// TwinCAT 3 PLC project DAS_assignment1_AbhijitDas
// ProgramVersion: 3.1.0.9
// libraries:
//   Standard, * (System)
//   VisuElem3DPath, 3.5.6.0 (System)
//   VisuElemMeter, 3.5.6.0 (System)
//   VisuElems, 3.5.6.10 (System)
//   VisuElemsDateTime, 3.5.6.0 (System)
//   VisuElemsSpecialControls, 3.5.6.0 (System)
//   VisuElemsWinControls, 3.5.6.0 (System)
//   VisuElemTextEditor, 3.5.6.0 (System)
//   visuinputs, 3.5.6.0 (system)
//   VisuNativeControl, 3.5.6.0 (System)
//   Tc2_Standard, * (Beckhoff Automation GmbH)
//   Tc2_System, * (Beckhoff Automation GmbH)
//   Tc3_Interfaces, * (Beckhoff Automation GmbH)
//   Tc3_Module, * (Beckhoff Automation GmbH)
//   VisuDialogs, * (System)
// project tree:
//   / GlobalTextList.TcGTLO, GVL.TcGVL, PlcTask.TcTTO, Visualization Manager.TcVMO (not stored)
//   POUs/ DistStationSensors.TcPOU, DistStationControl.TcPOU, MAIN.TcPOU, TestStationControl.TcPOU, TestStationSensors.TcPOU
//   VISUs/ StationVisualProgram.TcPOU, StationVisual.TcVIS

CONFIGURATION DAS_assignment1_AbhijitDas
    RESOURCE PLC ON TwinCAT3
        TASK PlcTask(INTERVAL := T#10ms, PRIORITY := 20);
        PROGRAM MAIN WITH PlcTask : MAIN;
    END_RESOURCE
END_CONFIGURATION

// ---- GVL.TcGVL
VAR_GLOBAL
	
	
	insertMag: BOOL; (* Variable for inserting Cylinder base in the stack magazine barrel*)
	Check_Mat: BOOL; (* Variable for starting the material checking actuator*)
	H_Meas: BOOL;   (* Variable for starting the height measurement actuator*)
	Testing: BOOL;  (* Variable that is set while the testing station is busy*)
	T_reset: TIME;	(* time to imitate reset value*)
	VisuReset: BOOL := TRUE; (* Variable is used to reset the visualization when reset is pressed*)
	forVisuPos5: BOOL;   (* used for visual only*)
	
	
	(* These variables are all as described in the provided MPS Festo documents*)
	start: BOOL;
	stop: BOOL;
	reset: BOOL;
	Mag: BOOL;
	Mag_back: BOOL := TRUE;
	Mag_front: BOOL;
	Vacuum: BOOL;
	Arm_take: BOOL := TRUE;
	Arm_put: BOOL;
	Mat_sen: BOOL;
	Vacumon: BOOL;
	Vacumoff: BOOL;
	Armleft: BOOL;
	Armright: BOOL;
	Auto: BOOL;
	Automan: BOOL;
	L_START: BOOL;
	L_RESET: BOOL;
	LiftDown: BOOL;
	MatPush: BOOL;
	Slide: BOOL;
	Part_AV: BOOL;
	Lift_Up: BOOL;
	Push_Ba: BOOL;
	Sen_Mat: BOOL;
	LiftUp: BOOL;
	Lift_Down: BOOL := TRUE;
	Work_ok: BOOL := TRUE;
	Follow: BOOL;
	Safety_barrier: BOOL;
	
	
END_VAR

// ---- POUs/MAIN.TcPOU
PROGRAM MAIN
VAR
END_VAR

DistStationSensors();
DistStationControl();
TestStationSensors();
TestStationControl();
StationVisualProgram();

END_PROGRAM

// ---- POUs/DistStationSensors.TcPOU
PROGRAM DistStationSensors
VAR
	StackLimit: WORD := 8; (* Stating the limit of the stack module barrel*)
	null: BOOL; (* set when stack module barrel is empty*)
	Current: WORD ; (* Current number of base/s in the stack module barrel*)
	LimitReached: BOOL; (* set when the stack module barrel is full*)
	counter1: CTUD;  (* counter used to count the number of bases inserted in the barrel*)
	
END_VAR
VAR // added by the converter: edge detectors and wires of the graphical bodies
    _w1, _w2, _w3, _w4 : BOOL;
END_VAR

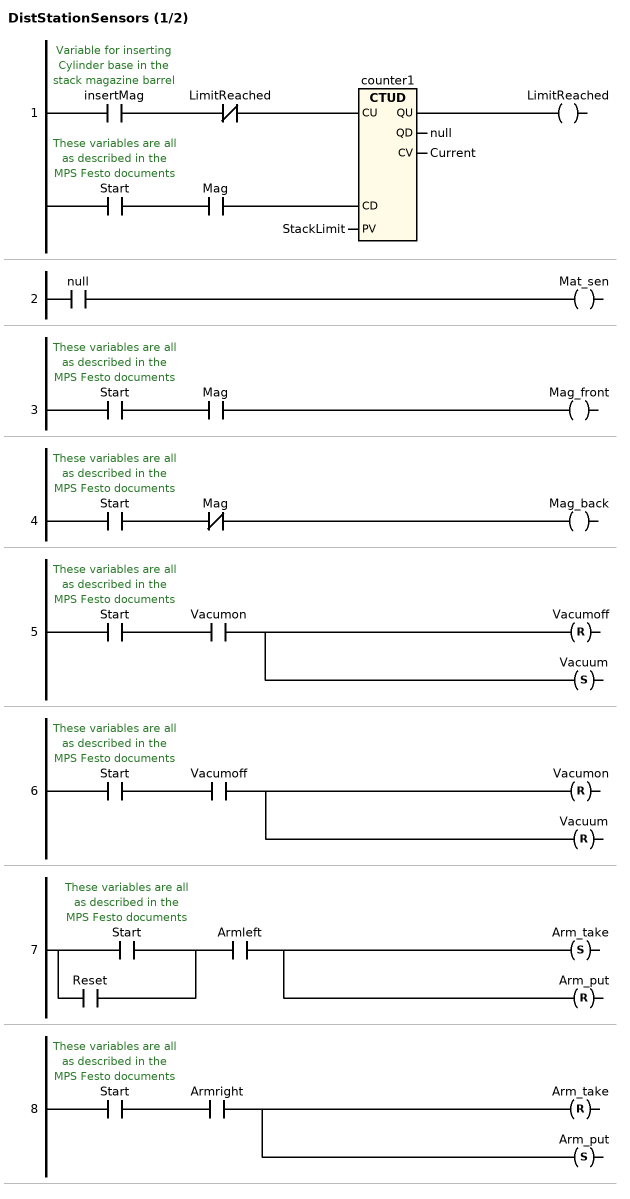
// NETWORK 1
//   insertMag: Variable for inserting Cylinder base in the stack magazine barrel
//   Start: These variables are all as described in the MPS Festo documents
counter1(
    CU := insertMag AND NOT LimitReached,
    CD := Start AND Mag,
    PV := StackLimit,
    QD => null,
    CV => Current); // CTUD
LimitReached := counter1.QU;

// NETWORK 2
Mat_sen := null;

// NETWORK 3
//   Start: These variables are all as described in the MPS Festo documents
Mag_front := Start AND Mag;

// NETWORK 4
//   Start: These variables are all as described in the MPS Festo documents
Mag_back := Start AND NOT Mag;

// NETWORK 5
//   Start: These variables are all as described in the MPS Festo documents
_w1 := Start AND Vacumon;
Vacumoff R= _w1;
Vacuum S= _w1;

// NETWORK 6
//   Start: These variables are all as described in the MPS Festo documents
_w2 := Start AND Vacumoff;
Vacumon R= _w2;
Vacuum R= _w2;

// NETWORK 7
//   Start: These variables are all as described in the MPS Festo documents
_w3 := (Start OR Reset) AND Armleft;
Arm_take S= _w3;
Arm_put R= _w3;

// NETWORK 8
//   Start: These variables are all as described in the MPS Festo documents
_w4 := Start AND Armright;
Arm_take R= _w4;
Arm_put S= _w4;

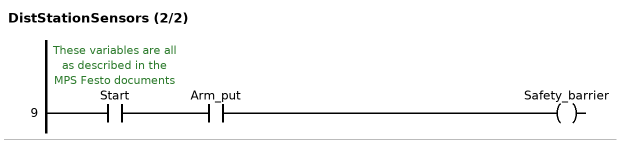
// NETWORK 9
//   Start: These variables are all as described in the MPS Festo documents
Safety_barrier := Start AND Arm_put;

END_PROGRAM

// ---- POUs/DistStationControl.TcPOU
PROGRAM DistStationControl
VAR
	(* These timers are used to imitate the moving time in the visualization*)
	T1: TIME := TIME#1S0MS;
	T2: TIME := TIME#2000MS;
	TON1: TON;
	TON2: TON;
	TON3: TON;
	TON4: TON;
	TON5: TON;
	TON6: TON;
	
	
	InReset: BOOL; (*  Variable for knowing whether the system is already in reset*)
	
	(* These are just used to maintain the sequence or flow*)
	next1: BOOL;
	next2: BOOL;
END_VAR
VAR // added by the converter: edge detectors and wires of the graphical bodies
    _w1, _w2 : BOOL;
END_VAR

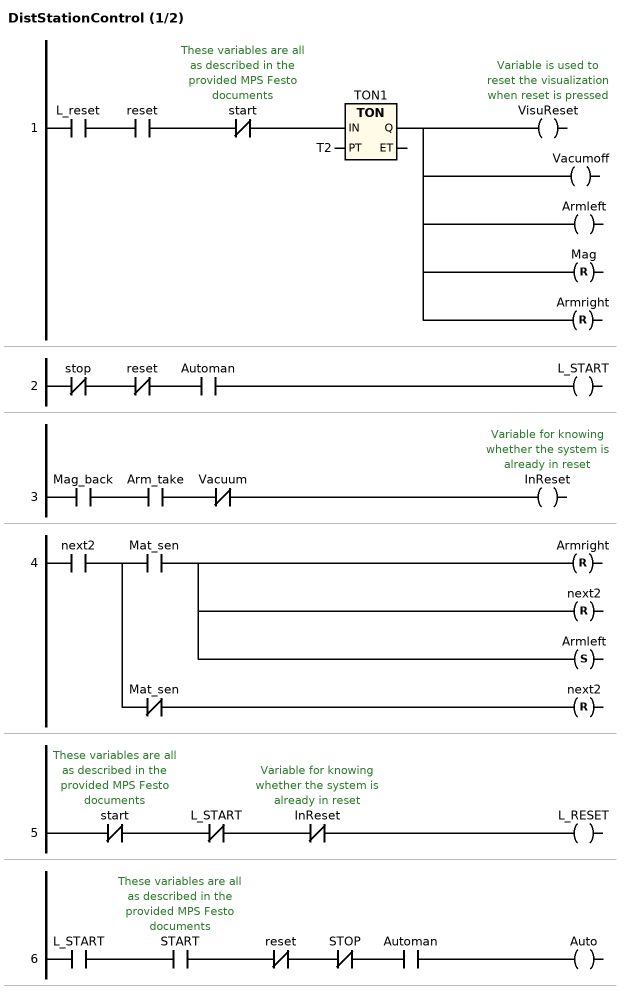
// NETWORK 1
//   start: These variables are all as described in the provided MPS Festo documents
//   VisuReset: Variable is used to reset the visualization when reset is pressed
TON1(IN := L_reset AND reset AND NOT start, PT := T2); // TON
VisuReset := TON1.Q;
Vacumoff := TON1.Q;
Armleft := TON1.Q;
Mag R= TON1.Q;
Armright R= TON1.Q;

// NETWORK 2
L_START := NOT stop AND NOT reset AND Automan;

// NETWORK 3
//   InReset: Variable for knowing whether the system is already in reset
InReset := Mag_back AND Arm_take AND NOT Vacuum;

// NETWORK 4
_w1 := next2;
_w2 := _w1 AND Mat_sen;
Armright R= _w2;
next2 R= _w2;
Armleft S= _w2;
next2 R= _w1 AND NOT Mat_sen;

// NETWORK 5
//   start: These variables are all as described in the provided MPS Festo documents
//   InReset: Variable for knowing whether the system is already in reset
L_RESET := NOT start AND NOT L_START AND NOT InReset;

// NETWORK 6
//   START: These variables are all as described in the provided MPS Festo documents
Auto := (L_START AND START AND NOT reset AND NOT STOP) AND Automan;

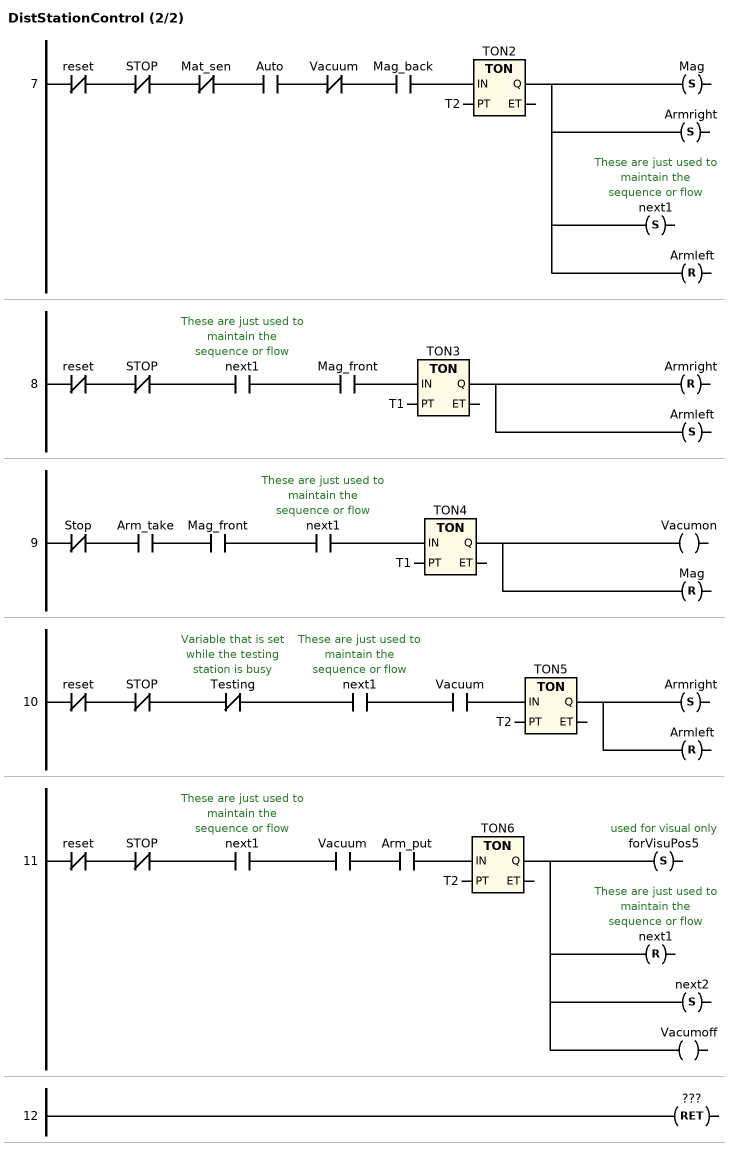
// NETWORK 7
//   next1: These are just used to maintain the sequence or flow
TON2(IN := NOT reset AND NOT STOP AND NOT Mat_sen AND Auto AND NOT Vacuum AND Mag_back, PT := T2); // TON
Mag S= TON2.Q;
Armright S= TON2.Q;
next1 S= TON2.Q;
Armleft R= TON2.Q;

// NETWORK 8
//   next1: These are just used to maintain the sequence or flow
//   T1: These timers are used to imitate the moving time in the visualization
TON3(IN := NOT reset AND NOT STOP AND next1 AND Mag_front, PT := T1); // TON
Armright R= TON3.Q;
Armleft S= TON3.Q;

// NETWORK 9
//   next1: These are just used to maintain the sequence or flow
//   T1: These timers are used to imitate the moving time in the visualization
TON4(IN := NOT Stop AND Arm_take AND Mag_front AND next1, PT := T1); // TON
Vacumon := TON4.Q;
Mag R= TON4.Q;

// NETWORK 10
//   Testing: Variable that is set while the testing station is busy
//   next1: These are just used to maintain the sequence or flow
TON5(IN := NOT reset AND NOT STOP AND NOT Testing AND next1 AND Vacuum, PT := T2); // TON
Armright S= TON5.Q;
Armleft R= TON5.Q;

// NETWORK 11
//   next1: These are just used to maintain the sequence or flow
//   forVisuPos5: used for visual only
TON6(IN := NOT reset AND NOT STOP AND next1 AND Vacuum AND Arm_put, PT := T2); // TON
forVisuPos5 S= TON6.Q;
next1 R= TON6.Q;
next2 S= TON6.Q;
Vacumoff := TON6.Q;

// NETWORK 12
RETURN;

END_PROGRAM

// ---- POUs/TestStationSensors.TcPOU
PROGRAM TestStationSensors
VAR
	(* These timers are used to imitate the moving time in the visualization*)
	t1: TIME := TIME#500MS;
	TON_0: TON;
	TON_1: TON;
	
END_VAR
VAR // added by the converter: edge detectors and wires of the graphical bodies
    _w1, _w2 : BOOL;
END_VAR

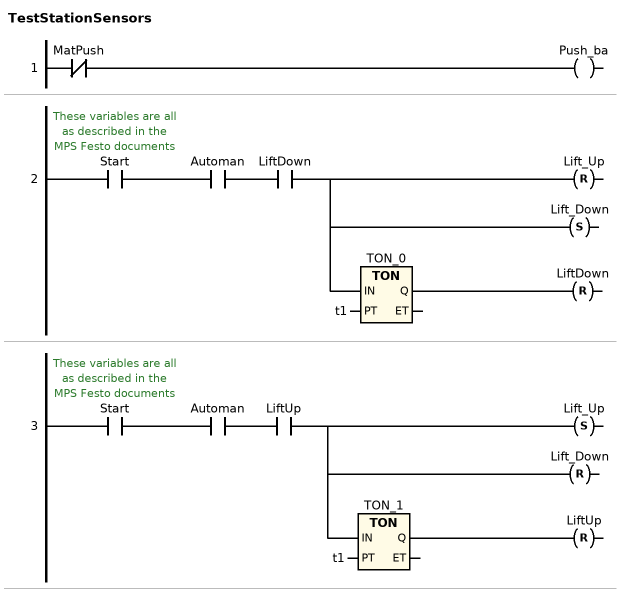
// NETWORK 1
Push_ba := NOT MatPush;

// NETWORK 2
//   Start: These variables are all as described in the MPS Festo documents
_w1 := Start AND Automan AND LiftDown;
Lift_Up R= _w1;
Lift_Down S= _w1;
TON_0(IN := _w1, PT := t1); // TON
LiftDown R= TON_0.Q;

// NETWORK 3
//   Start: These variables are all as described in the MPS Festo documents
_w2 := Start AND Automan AND LiftUp;
Lift_Up S= _w2;
Lift_Down R= _w2;
TON_1(IN := _w2, PT := t1); // TON
LiftUp R= TON_1.Q;

END_PROGRAM

// ---- POUs/TestStationControl.TcPOU
PROGRAM TestStationControl
VAR
	(* These timers are used to imitate the moving time in the visualization*)
	T_Mat_Check: TIME := TIME#2S0MS;
	T1: TIME := TIME#2S0MS;
	T_liftDown: TIME := TIME#2S0MS;
	T_H_meas: TIME := TIME#2S0MS;
	T_MatPush: TIME := TIME#1S0MS;
	TON_Mat_Check: TON;
	TON_MatPush: TON;
	TON_MatPush2: TON;
	TON_Lift: TON;
	TON1: TON;
	TON_0: TON;
	TON_1: TON;
	TON_2: TON;
	TON_H_Meas: TON;
	TON_Lift2: TON;
	TON_reset: TON;
	
	(* These are just used to maintain the sequence or flow*)
	next2: BOOL;
	next3: BOOL;
	next4: BOOL;
END_VAR
VAR // added by the converter: edge detectors and wires of the graphical bodies
    _w1, _w2, _w3, _w4, _w5, _w6, _w7 : BOOL;
END_VAR

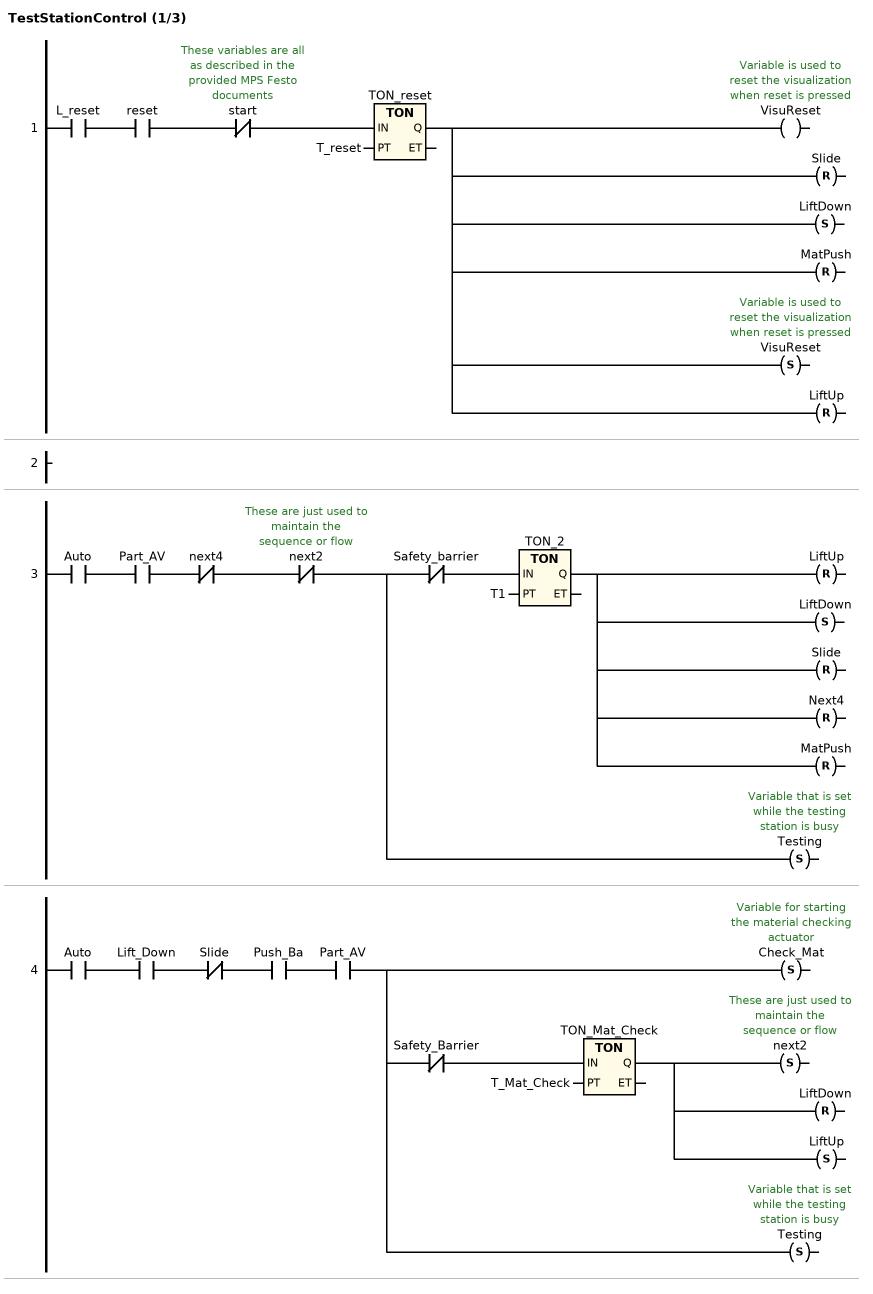
// NETWORK 1
//   start: These variables are all as described in the provided MPS Festo documents
//   T_reset: time to imitate reset value
//   VisuReset: Variable is used to reset the visualization when reset is pressed
TON_reset(IN := L_reset AND reset AND NOT start, PT := T_reset); // TON
VisuReset := TON_reset.Q;
Slide R= TON_reset.Q;
LiftDown S= TON_reset.Q;
MatPush R= TON_reset.Q;
VisuReset S= TON_reset.Q;
LiftUp R= TON_reset.Q;

// NETWORK 2

// NETWORK 3
//   next2: These are just used to maintain the sequence or flow
//   Testing: Variable that is set while the testing station is busy
_w1 := Auto AND Part_AV AND NOT next4 AND NOT next2;
TON_2(IN := _w1 AND NOT Safety_barrier, PT := T1); // TON
LiftUp R= TON_2.Q;
LiftDown S= TON_2.Q;
Slide R= TON_2.Q;
Next4 R= TON_2.Q;
MatPush R= TON_2.Q;
Testing S= _w1;

// NETWORK 4
//   Check_Mat: Variable for starting the material checking actuator
//   T_Mat_Check: These timers are used to imitate the moving time in the visualization
//   next2: These are just used to maintain the sequence or flow
//   Testing: Variable that is set while the testing station is busy
_w2 := Auto AND Lift_Down AND NOT Slide AND Push_Ba AND Part_AV;
Check_Mat S= _w2;
TON_Mat_Check(IN := _w2 AND NOT Safety_Barrier, PT := T_Mat_Check); // TON
next2 S= TON_Mat_Check.Q;
LiftDown R= TON_Mat_Check.Q;
LiftUp S= TON_Mat_Check.Q;
Testing S= _w2;

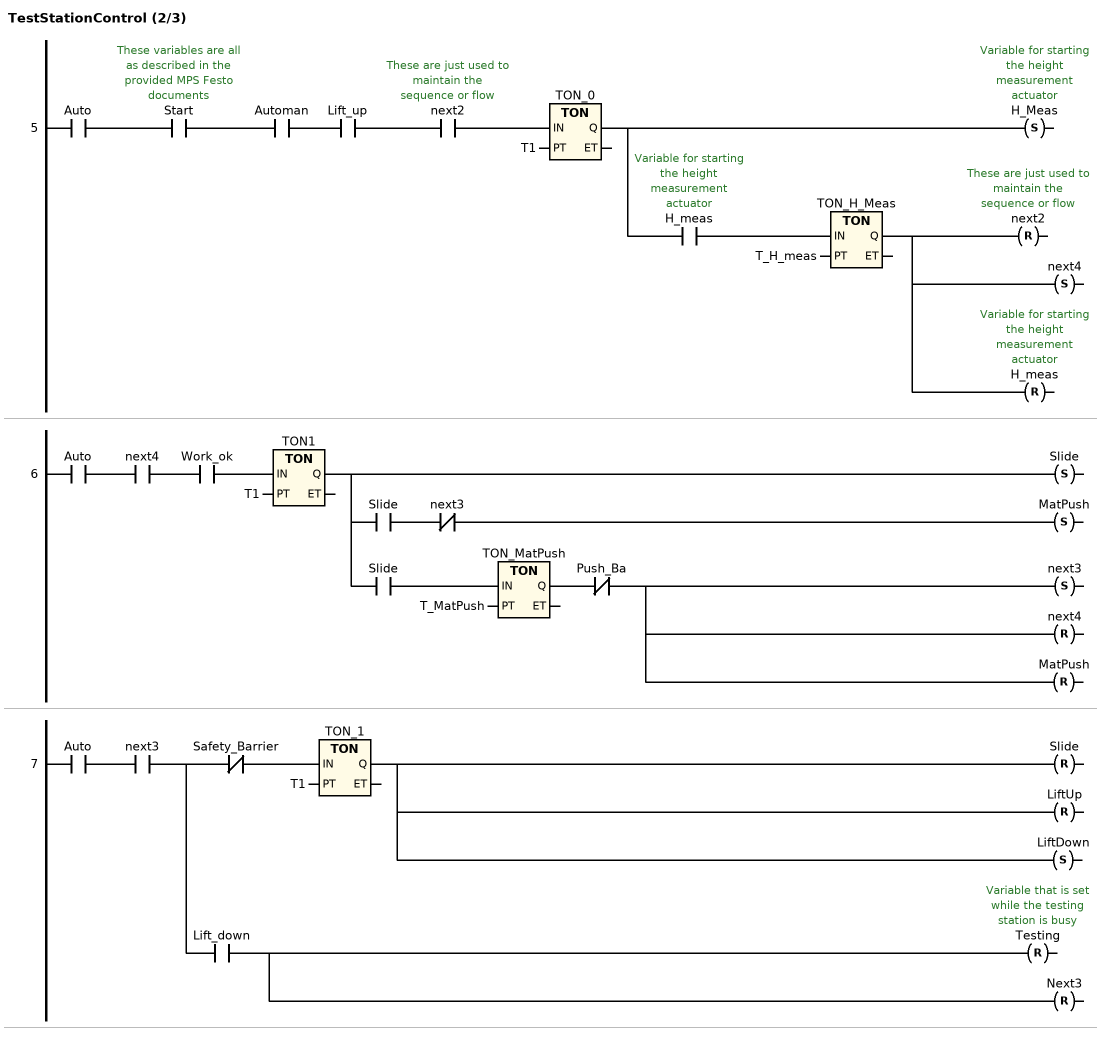
// NETWORK 5
//   Start: These variables are all as described in the provided MPS Festo documents
//   next2: These are just used to maintain the sequence or flow
//   H_Meas: Variable for starting the height measurement actuator
//   H_meas: Variable for starting the height measurement actuator
TON_0(IN := Auto AND Start AND Automan AND Lift_up AND next2, PT := T1); // TON
H_Meas S= TON_0.Q;
TON_H_Meas(IN := TON_0.Q AND H_meas, PT := T_H_meas); // TON
next2 R= TON_H_Meas.Q;
next4 S= TON_H_Meas.Q;
H_meas R= TON_H_Meas.Q;

// NETWORK 6
TON1(IN := Auto AND next4 AND Work_ok, PT := T1); // TON
Slide S= TON1.Q;
MatPush S= TON1.Q AND Slide AND NOT next3;
TON_MatPush(IN := TON1.Q AND Slide, PT := T_MatPush); // TON
_w3 := TON_MatPush.Q AND NOT Push_Ba;
next3 S= _w3;
next4 R= _w3;
MatPush R= _w3;

// NETWORK 7
//   Testing: Variable that is set while the testing station is busy
_w4 := Auto AND next3;
TON_1(IN := _w4 AND NOT Safety_Barrier, PT := T1); // TON
Slide R= TON_1.Q;
LiftUp R= TON_1.Q;
LiftDown S= TON_1.Q;
_w5 := _w4 AND Lift_down;
Testing R= _w5;
Next3 R= _w5;

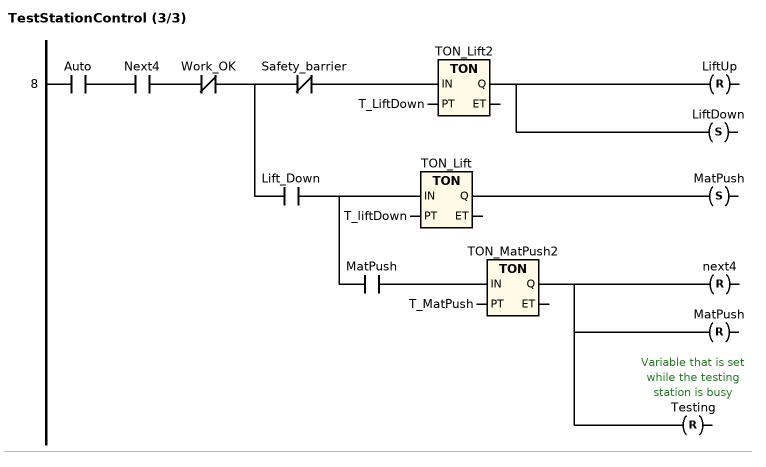
// NETWORK 8
//   Testing: Variable that is set while the testing station is busy
_w6 := Auto AND Next4 AND NOT Work_OK;
TON_Lift2(IN := _w6 AND NOT Safety_barrier, PT := T_LiftDown); // TON
LiftUp R= TON_Lift2.Q;
LiftDown S= TON_Lift2.Q;
_w7 := _w6 AND Lift_Down;
TON_Lift(IN := _w7, PT := T_liftDown); // TON
MatPush S= TON_Lift.Q;
TON_MatPush2(IN := _w7 AND MatPush, PT := T_MatPush); // TON
next4 R= TON_MatPush2.Q;
MatPush R= TON_MatPush2.Q;
Testing R= TON_MatPush2.Q;

END_PROGRAM

// ---- VISUs/StationVisualProgram.TcPOU
PROGRAM StationVisualProgram
VAR
	
	
	(* These are all used for animating the different positions of the cylinder bases *)
	MagPos1: BOOL := TRUE;
	MagPos2: BOOL := TRUE;
	MagPos3: BOOL := TRUE;
	MagPos4: BOOL := TRUE;
	MagPos5: BOOL := TRUE;
	BasePos6: BOOL := TRUE;
	BasePos7: BOOL :=  TRUE;
	BasePos7a: BOOL := TRUE;
	BasePos7b: BOOL := TRUE;
	BasePos7c: BOOL := TRUE;
	BasePos7d: BOOL := TRUE;
	BasePos7e: BOOL := TRUE;
	BasePos8: BOOL := TRUE;
	BasePos8a: BOOL := TRUE;
	BasePos8b: BOOL := TRUE;
	
	(*Used to animate the pusher of the testing station*)
	EjecCylDown: BOOL := TRUE;
	EjecCylUp: BOOL := TRUE;
	
	(* These timers are used to imitate the moving time in the visualization*)
	T_hMeas: TIME := TIME#1S500MS;
	t_half: TIME := TIME#250MS;
	TON_0: TON;
	TON_1: TON;
	TON_2: TON;
	TON_3: TON;
	TON_4: TON;
	TON_5: TON;
	TON_6: TON;
	TON_7: TON;
	TON_8: TON;
	TON_9: TON;
	
	(* These are just used to maintain the sequence or flow*)
	keep1: BOOL;
	next2: BOOL;
	Next3: BOOL;	
	Dummy: BOOL;
	
	H_MeasCylDo: BOOL := TRUE; (*Used to animate the measuring actuator*)
	
END_VAR
VAR // added by the converter: edge detectors and wires of the graphical bodies
    _w1, _w2, _w3, _w4, _w5, _w6, _w7, _w8, _w9, _w10, _w11, _w12, _w13, _w14, _w15, _w16, _w17, _w18, _w19, _w20 : BOOL;
END_VAR

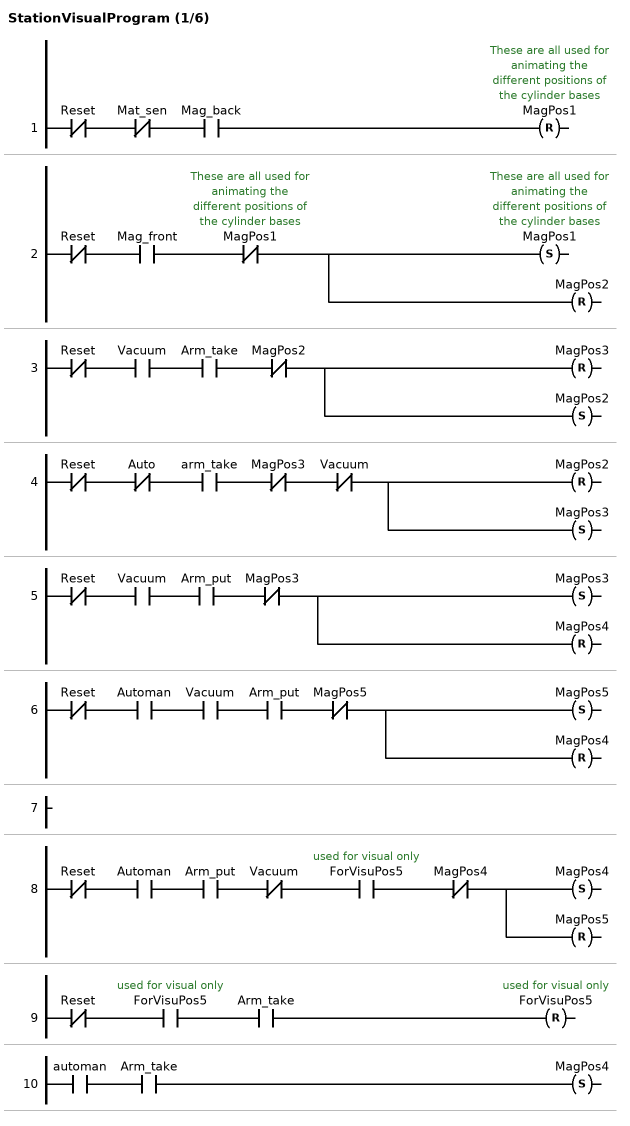
// NETWORK 1
//   MagPos1: These are all used for animating the different positions of the cylinder bases
MagPos1 R= NOT Reset AND NOT Mat_sen AND Mag_back;

// NETWORK 2
//   MagPos1: These are all used for animating the different positions of the cylinder bases
_w1 := NOT Reset AND Mag_front AND NOT MagPos1;
MagPos1 S= _w1;
MagPos2 R= _w1;

// NETWORK 3
_w2 := NOT Reset AND Vacuum AND Arm_take AND NOT MagPos2;
MagPos3 R= _w2;
MagPos2 S= _w2;

// NETWORK 4
_w3 := NOT Reset AND NOT Auto AND arm_take AND NOT MagPos3 AND NOT Vacuum;
MagPos2 R= _w3;
MagPos3 S= _w3;

// NETWORK 5
_w4 := NOT Reset AND Vacuum AND Arm_put AND NOT MagPos3;
MagPos3 S= _w4;
MagPos4 R= _w4;

// NETWORK 6
_w5 := NOT Reset AND Automan AND Vacuum AND Arm_put AND NOT MagPos5;
MagPos5 S= _w5;
MagPos4 R= _w5;

// NETWORK 7

// NETWORK 8
//   ForVisuPos5: used for visual only
_w6 := NOT Reset AND Automan AND Arm_put AND NOT Vacuum AND ForVisuPos5 AND NOT MagPos4;
MagPos4 S= _w6;
MagPos5 R= _w6;

// NETWORK 9
//   ForVisuPos5: used for visual only
ForVisuPos5 R= NOT Reset AND ForVisuPos5 AND Arm_take;

// NETWORK 10
MagPos4 S= automan AND Arm_take;

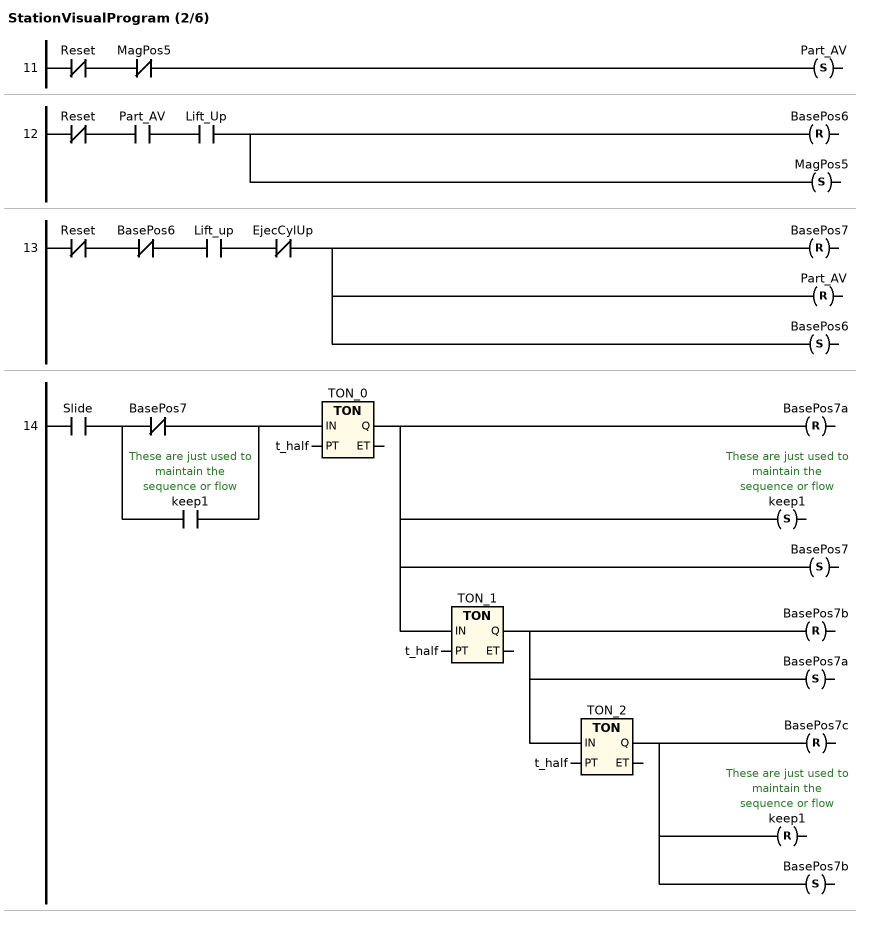
// NETWORK 11
Part_AV S= NOT Reset AND NOT MagPos5;

// NETWORK 12
_w7 := NOT Reset AND Part_AV AND Lift_Up;
BasePos6 R= _w7;
MagPos5 S= _w7;

// NETWORK 13
_w8 := NOT Reset AND NOT BasePos6 AND Lift_up AND NOT EjecCylUp;
BasePos7 R= _w8;
Part_AV R= _w8;
BasePos6 S= _w8;

// NETWORK 14
//   keep1: These are just used to maintain the sequence or flow
TON_0(IN := Slide AND (NOT BasePos7 OR keep1), PT := t_half); // TON
BasePos7a R= TON_0.Q;
keep1 S= TON_0.Q;
BasePos7 S= TON_0.Q;
TON_1(IN := TON_0.Q, PT := t_half); // TON
BasePos7b R= TON_1.Q;
BasePos7a S= TON_1.Q;
TON_2(IN := TON_1.Q, PT := t_half); // TON
BasePos7c R= TON_2.Q;
keep1 R= TON_2.Q;
BasePos7b S= TON_2.Q;

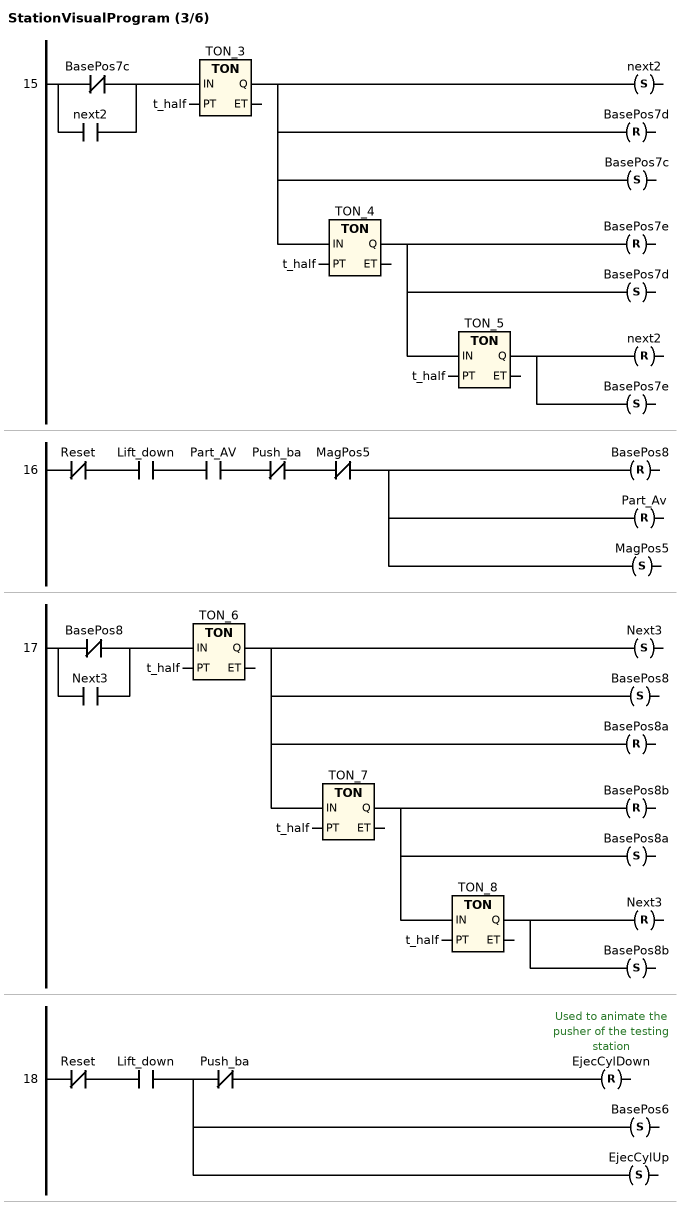
// NETWORK 15
TON_3(IN := NOT BasePos7c OR next2, PT := t_half); // TON
next2 S= TON_3.Q;
BasePos7d R= TON_3.Q;
BasePos7c S= TON_3.Q;
TON_4(IN := TON_3.Q, PT := t_half); // TON
BasePos7e R= TON_4.Q;
BasePos7d S= TON_4.Q;
TON_5(IN := TON_4.Q, PT := t_half); // TON
next2 R= TON_5.Q;
BasePos7e S= TON_5.Q;

// NETWORK 16
_w9 := NOT Reset AND Lift_down AND Part_AV AND NOT Push_ba AND NOT MagPos5;
BasePos8 R= _w9;
Part_Av R= _w9;
MagPos5 S= _w9;

// NETWORK 17
TON_6(IN := NOT BasePos8 OR Next3, PT := t_half); // TON
Next3 S= TON_6.Q;
BasePos8 S= TON_6.Q;
BasePos8a R= TON_6.Q;
TON_7(IN := TON_6.Q, PT := t_half); // TON
BasePos8b R= TON_7.Q;
BasePos8a S= TON_7.Q;
TON_8(IN := TON_7.Q, PT := t_half); // TON
Next3 R= TON_8.Q;
BasePos8b S= TON_8.Q;

// NETWORK 18
//   EjecCylDown: Used to animate the pusher of the testing station
_w10 := NOT Reset AND Lift_down;
EjecCylDown R= _w10 AND NOT Push_ba;
BasePos6 S= _w10;
EjecCylUp S= _w10;

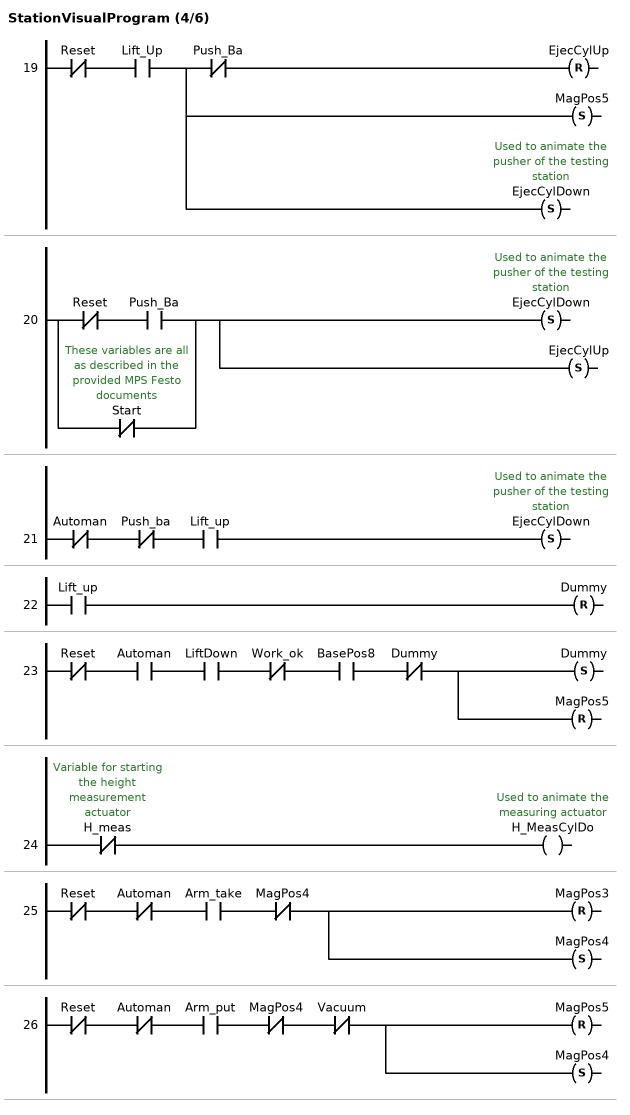
// NETWORK 19
//   EjecCylDown: Used to animate the pusher of the testing station
_w11 := NOT Reset AND Lift_Up;
EjecCylUp R= _w11 AND NOT Push_Ba;
MagPos5 S= _w11;
EjecCylDown S= _w11;

// NETWORK 20
//   Start: These variables are all as described in the provided MPS Festo documents
//   EjecCylDown: Used to animate the pusher of the testing station
_w12 := NOT Reset AND Push_Ba OR NOT Start;
EjecCylDown S= _w12;
EjecCylUp S= _w12;

// NETWORK 21
//   EjecCylDown: Used to animate the pusher of the testing station
EjecCylDown S= NOT Automan AND NOT Push_ba AND Lift_up;

// NETWORK 22
Dummy R= Lift_up;

// NETWORK 23
_w13 := NOT Reset AND Automan AND LiftDown AND NOT Work_ok AND BasePos8 AND NOT Dummy;
Dummy S= _w13;
MagPos5 R= _w13;

// NETWORK 24
//   H_meas: Variable for starting the height measurement actuator
//   H_MeasCylDo: Used to animate the measuring actuator
H_MeasCylDo := NOT H_meas;

// NETWORK 25
_w14 := NOT Reset AND NOT Automan AND Arm_take AND NOT MagPos4;
MagPos3 R= _w14;
MagPos4 S= _w14;

// NETWORK 26
_w15 := NOT Reset AND NOT Automan AND Arm_put AND NOT MagPos4 AND NOT Vacuum;
MagPos5 R= _w15;
MagPos4 S= _w15;

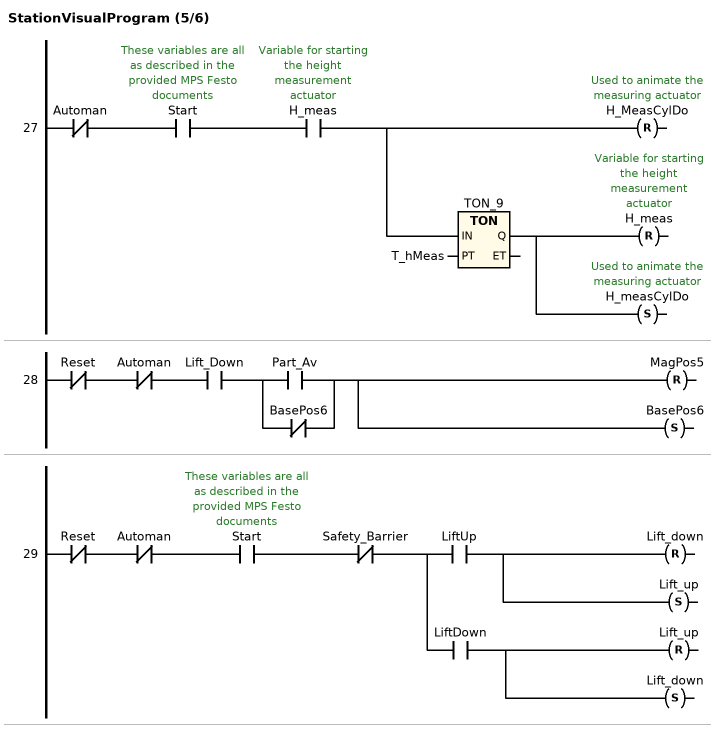
// NETWORK 27
//   Start: These variables are all as described in the provided MPS Festo documents
//   H_meas: Variable for starting the height measurement actuator
//   H_MeasCylDo: Used to animate the measuring actuator
//   T_hMeas: These timers are used to imitate the moving time in the visualization
//   H_measCylDo: Used to animate the measuring actuator
_w16 := NOT Automan AND Start AND H_meas;
H_MeasCylDo R= _w16;
TON_9(IN := _w16, PT := T_hMeas); // TON
H_meas R= TON_9.Q;
H_measCylDo S= TON_9.Q;

// NETWORK 28
_w17 := NOT Reset AND NOT Automan AND Lift_Down AND (Part_Av OR NOT BasePos6);
MagPos5 R= _w17;
BasePos6 S= _w17;

// NETWORK 29
//   Start: These variables are all as described in the provided MPS Festo documents
_w18 := NOT Reset AND NOT Automan AND Start AND NOT Safety_Barrier;
_w19 := _w18 AND LiftUp;
Lift_down R= _w19;
Lift_up S= _w19;
_w20 := _w18 AND LiftDown;
Lift_up R= _w20;
Lift_down S= _w20;

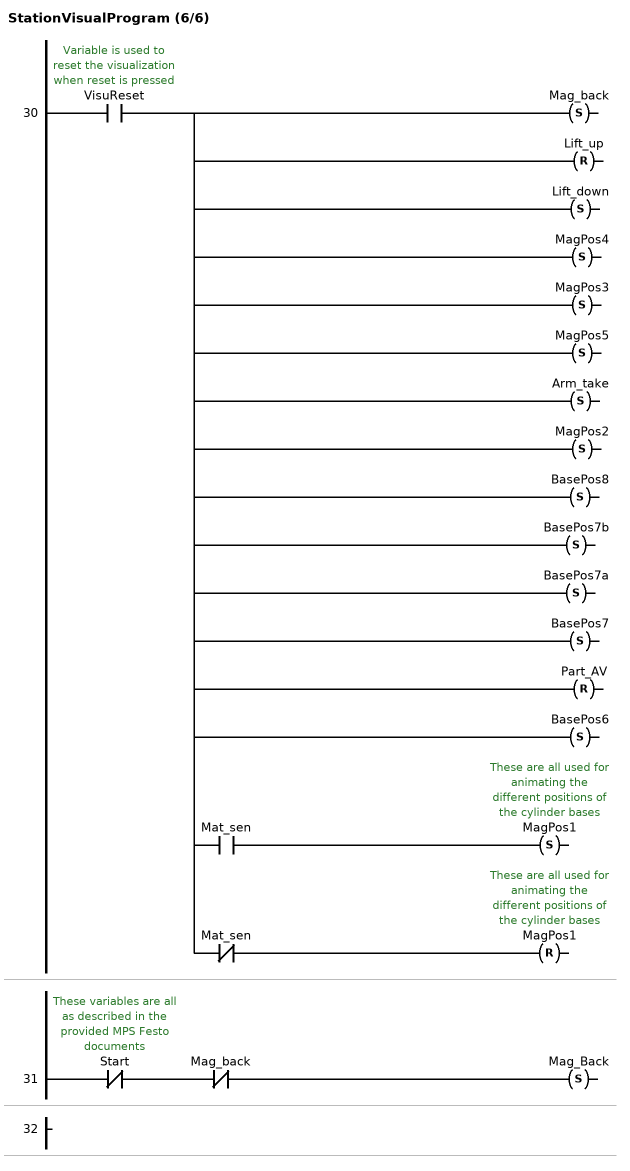
// NETWORK 30
//   VisuReset: Variable is used to reset the visualization when reset is pressed
//   MagPos1: These are all used for animating the different positions of the cylinder bases
Mag_back S= VisuReset;
Lift_up R= VisuReset;
Lift_down S= VisuReset;
MagPos4 S= VisuReset;
MagPos3 S= VisuReset;
MagPos5 S= VisuReset;
Arm_take S= VisuReset;
MagPos2 S= VisuReset;
BasePos8 S= VisuReset;
BasePos7b S= VisuReset;
BasePos7a S= VisuReset;
BasePos7 S= VisuReset;
Part_AV R= VisuReset;
BasePos6 S= VisuReset;
MagPos1 S= VisuReset AND Mat_sen;
MagPos1 R= VisuReset AND NOT Mat_sen;

// NETWORK 31
//   Start: These variables are all as described in the provided MPS Festo documents
Mag_Back S= NOT Start AND NOT Mag_back;

// NETWORK 32

END_PROGRAM

// ---- GlobalTextList.TcGTLO
TEXTLIST GlobalTextList
  1 = '77'
  32 = 'Air Slider On/Off'
  22 = 'Arm Left'
  26 = 'ARM LEFT'
  21 = 'Arm Left/ Right'
  24 = 'ARM Right'
  25 = 'ARM RIGHT'
  23 = 'ARMAArm'
  11 = 'AUTO/Manual'
  4 = 'automan'
  43 = 'Automated Control'
  46 = 'Base 1'
  47 = 'Base 2'
  48 = 'Base 3'
  49 = 'Base 4'
  50 = 'Base 5'
  51 = 'Base 6'
  52 = 'Base 7'
  14 = 'Distribution Station Control'
  18 = 'Ejectory Cylinder'
  28 = 'Ejectory Cylinder  front'
  27 = 'Ejectory Cylinder  front/'
  19 = 'Ejectory Cylinder  front/ back'
  37 = 'Ejectory Cylinder  front/back'
  29 = 'Ejectory Cylinder Back'
  39 = 'Height'
  41 = 'Height Not OK'
  40 = 'Height OK'
  42 = 'Imitiate Height Parameter'
  12 = 'Indicaotor 1'
  13 = 'Indicator 2'
  15 = 'Insert Mag'
  5 = 'InsertMag'
  31 = 'Lift Down'
  30 = 'Lift Up'
  2 = 'Loading Mag'
  6 = 'LoadMag'
  7 = 'looper'
  17 = 'Manual Control'
  59 = 'Manual Control: Turn AUTO OFF then press START  '
  45 = 'Measure Height'
  55 = 'PLEASE NOTE!!'
  57 = 'PLEASE NOTE!!   '
  56 = 'PLEASE NOTE!!   To RESET the system, STOP button must first be pressed. To manually control, press START with AUTO turned off. '
  33 = 'Pushing Cylinder Back'
  38 = 'Pushing Cylinder Back/ Front'
  34 = 'Pushing Cylinder Front'
  44 = 'Put Cylinder Base'
  54 = 'REJECTED :('
  53 = 'REJECTED MAAL'
  10 = 'RESET'
  16 = 'Reset'
  3 = 'start'
  8 = 'START'
  9 = 'STOP'
  58 = 'To Reset: First press STOP then RESET '
  0 = 'ttt'
  36 = 'Vacuum Off'
  35 = 'Vacuum On'
  20 = 'Vacuum On/OFF'
END_TEXTLIST

// ---- VISUs/StationVisual.TcVIS
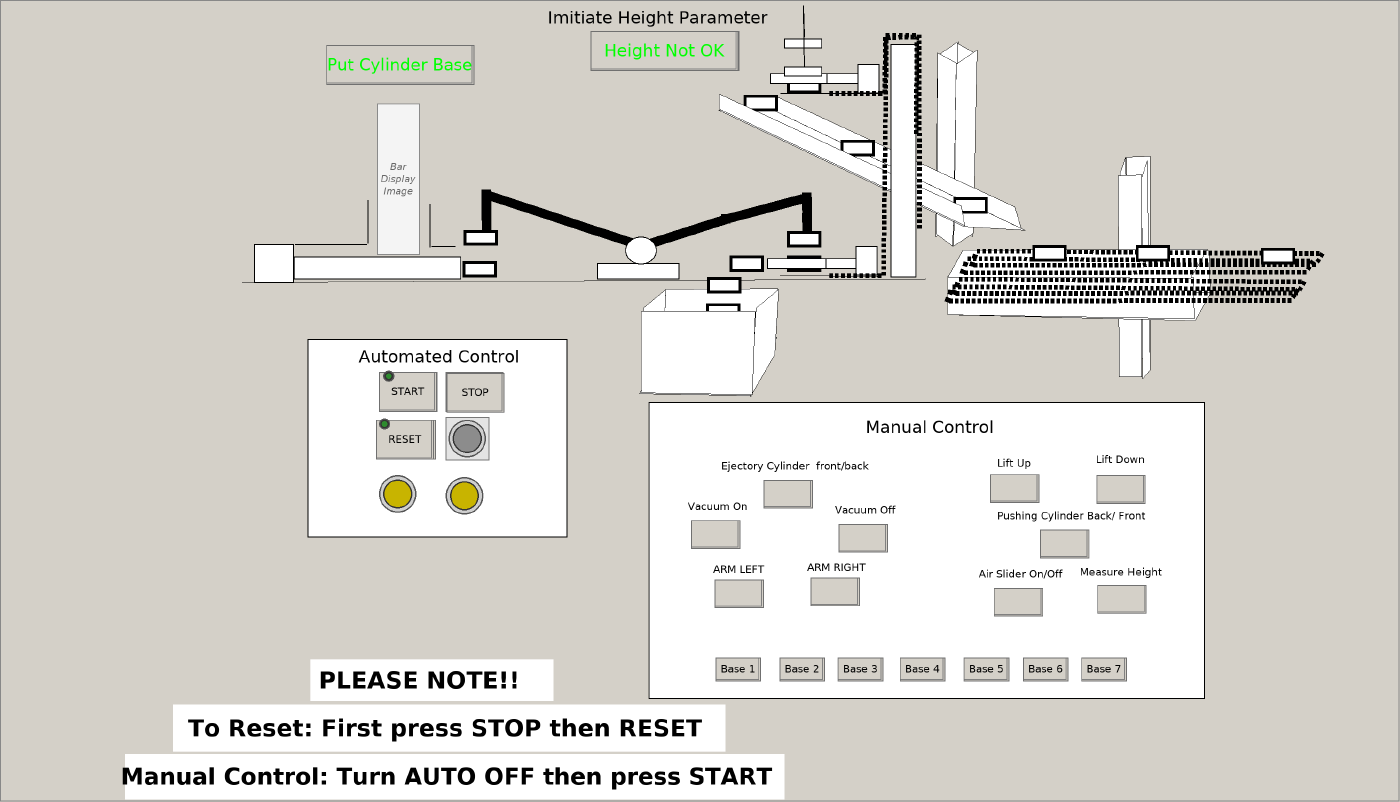
VISUALIZATION StationVisual  // 1489x854
    RoundedRectangle (837,272 36x17), invisible if: StationVisualProgram.MagPos5
    RoundedRectangle (816,275 105x11), invisible if: StationVisualProgram.EjecCylDown
    RoundedRectangle (837,82 36x17), invisible if: StationVisualProgram.BasePos6
    RoundedRectangle (819,78 105x11), invisible if: StationVisualProgram.EjecCylUp
    Polygon (684,328) (708,308) (706,360) (684,419)
    Polygon (708,308) (827,307) (824,362) (706,360)
    Polygon (707,359) (826,359) (798,421) (680,419)
    Polygon (804,328) (828,308) (824,377) (798,422)
    RoundedRectangle (751,323 36x17), invisible if: StationVisualProgram.BasePos8b
    Group (995,44 44x297)
        Polygon (0,208) (2,15) (24,0) (20,195)
        Polygon (22,195) (23,2) (43,13) (39,208)
        Polygon (19,218) (22,24) (44,9) (40,204)
        Polygon (1,205) (2,12) (22,23) (18,218)
    Polygon (764,117) (1025,241) (1090,245) (824,118)
    Polygon (822,117) (1086,243) (1079,220) (822,101)
    Group (1189,166 50x236)
        Polygon (3,233) (2,19) (8,1) (11,224)
        Polygon (10,215) (9,1) (34,0) (34,215)
        Polygon (1,235) (0,21) (25,20) (25,235)
        Polygon (26,237) (25,23) (31,5) (34,228)
    Polyline (680,261) (517,207) (517,217) (517,225) (517,230) (517,246), invisible if: Arm_put
    Polyline (685,261) (772,233) (858,210) (858,219) (858,232) (858,246), invisible if: Arm_take
    Rectangle (401,138 43x121), invisible if: RotDriveMag
    Line (391,229)
    Line (391,213) (391,259)
    Line (457,217) (457,263)
    Line (314,260) (390,260)
    Line (984,297) (258,301)
    Line (459,262) (484,262)
    Rectangle (287,273 106x24), invisible if: Mag_front
    RoundedRectangle (404,276 36x17), invisible if: StationVisualProgram.MagPos1
    RoundedRectangle (492,278 36x17), invisible if: StationVisualProgram.MagPos2
    BarDisplayImage (401,110 45x161), value: DistStationSensors.Current, style: BarDisplayImage-Gray, scale format: %.1f, scale 0..8
    Button (347,48 157x42), "Put Cylinder Base"
        tap insertMag
    Group (635,252 87x45)
        RoundedRectangle (0,28 87x17)
        Ellipse (30,0 33x29)
    RoundedRectangle (837,246 36x17), invisible if: StationVisualProgram.MagPos4
    RoundedRectangle (493,245 36x16), invisible if: StationVisualProgram.MagPos3
    Group (327,361 278x211)
        Rectangle (0,0 276x211)
        Group (147,35 50x28)
            Button (0,0 61x42), "STOP"
                toggle stop
            Button (1,1 61x42), "STOP", invisible if: stop
                toggle stop
        PushSwitchLed (142,83 56x46), tooltip "AUTO/Manual", variable: Automan, behaviour: TOGGLE, style: Switch-PushSwitchLed-Gray
        Lamp1 (68,142 56x46), tooltip "Indicaotor 1", variable: Mat_sen, style: Lamp-Lamp1-Yellow
        Lamp1 (139,144 56x46), tooltip "Indicator 2", style: Lamp-Lamp1-Yellow
        Label (2,7 276x24), "Automated Control"
        Group (76,35 50x28)
            Button (1,0 61x42), "START"
                toggle start
            Button (0,0 61x42), "START", invisible if: start
                toggle start
        Group (73,86 51x28)
            Button (2,0 61x42), "RESET"
                toggle reset
            Button (0,0 61x42), "RESET", invisible if: reset
                toggle reset
        Lamp1 (75,33 23x13), variable: L_START, style: Lamp-Lamp1-Green
        Lamp1 (72,84 20x13), variable: L_RESET, style: Lamp-Lamp1-Green
    Group (1008,265 479x76)
        Polygon (263,76) (1,70) (20,20) (281,44)
        Polygon (279,46) (17,42) (17,1) (278,2)
        Polygon (262,74) (0,70) (0,29) (261,30)
        Polygon (258,31) (0,30) (16,1) (276,0)
    Group (1007,267 476x30)
        Polyline (6,38) (373,41) (366,53) (0,54) (6,38)
        Polyline (13,30) (380,33) (373,45) (7,46) (13,30)
        Polyline (22,8) (389,11) (382,23) (16,24) (22,8)
        Polyline (32,0) (399,3) (392,15) (26,16) (32,0)
    RoundedRectangle (791,101 36x17), invisible if: StationVisualProgram.BasePos7
    RoundedRectangle (1098,261 36x17), invisible if: StationVisualProgram.BasePos7c
    RoundedRectangle (1208,261 36x17), invisible if: StationVisualProgram.BasePos7d
    RoundedRectangle (1341,264 36x17), invisible if: StationVisualProgram.BasePos7e
    RoundedRectangle (776,272 36x17), invisible if: StationVisualProgram.BasePos8
    RoundedRectangle (894,149 36x17), invisible if: StationVisualProgram.BasePos7a
    RoundedRectangle (1014,210 36x17), invisible if: StationVisualProgram.BasePos7b
    Group (878,262 55x31), invisible if: Lift_Up
        RoundedRectangle (0,13 50x11)
        RoundedRectangle (32,0 23x31)
    Group (879,68 56x31), invisible if: Lift_Down
        RoundedRectangle (0,10 50x11), invisible if: Lift_Down
        RoundedRectangle (33,0 23x31), invisible if: Lift_Down
    RoundedRectangle (752,295 36x17), invisible if: StationVisualProgram.BasePos8a
    Polygon (682,331) (803,331) (800,420) (682,418)
    Group (834,6 40x45), invisible if: H_Meas
        RoundedRectangle (0,35 40x10)
        Line (20,0) (21,33)
    Group (834,9 40x72), invisible if: StationVisualProgram.H_MeasCylDo
        Line (20,0) (21,66)
        RoundedRectangle (0,62 40x10)
    Rectangle (313,273 177x24), invisible if: Mag_back
    RoundedRectangle (270,260 42x41)
    Button (629,33 157x42), "Height OK"
        toggle Work_ok
    Button (628,33 157x42), "Height Not OK", invisible if: Work_ok
        toggle Work_ok
    Label (579,4 241x30), "Imitiate Height Parameter"
    Polygon (765,116) (1026,240) (1022,219) (765,100)
    RoundedRectangle (947,47 27x248)
    Group (830,39 145x255), invisible if: Lift_Up
        Polyline (52,254) (110,254) (113,1) (145,0) (144,106)
        Line (0,254) (103,255)
    Group (830,37 148x209), invisible if: Lift_Down
        Polyline (52,62) (111,62) (112,0) (147,0) (148,209)
        Line (0,62) (105,62)
    Rectangle (690,428 591x316)
    Label (851,443 276x24), "Manual Control"
    Group (676,509 175x75)
        Button (59,45 52x30)
            tap Vacumon
        Label (0,0 175x61), "Vacuum On"
    Group (698,576 175x71)
        Button (62,41 52x30)
            tap Armleft
        Label (0,0 175x61), "ARM LEFT"
    Group (802,574 175x71)
        Button (60,41 52x30)
            tap Armright
        Label (0,0 175x61), "ARM RIGHT"
    Group (758,466 175x75)
        Label (0,0 175x61), "Ejectory Cylinder front/back"
        Button (54,45 52x30), colour toggle: Mag
            toggle Mag
    Group (833,513 175x75)
        Button (59,45 52x30)
            tap Vacumoff
        Label (0,0 175x61), "Vacuum Off"
    Group (998,581 175x75)
        Button (59,45 52x30), colour toggle: Slide
            toggle Slide
        Label (0,0 175x61), "Air Slider On/Off"
    Group (991,463 175x72)
        Button (62,42 52x30)
            tap LiftUp
        Label (0,0 175x61), "Lift Up"
    Group (1104,459 175x77)
        Button (62,47 52x30)
            tap LiftDown
        Label (0,0 175x61), "Lift Down"
    Group (1052,519 175x75)
        Label (0,0 175x61), "Pushing Cylinder Back/ Front"
        Button (54,45 52x30)
            toggle MatPush
    Button (1167,623 52x30)
        toggle H_Meas
    Label (1105,579 175x61), "Measure Height"
    Button (761,700 48x25), "Base 1"
        toggle StationVisualProgram.MagPos1
    Button (829,700 48x25), "Base 2"
        toggle StationVisualProgram.MagPos2
    Button (891,700 48x25), "Base 3"
        toggle StationVisualProgram.MagPos3
    Button (957,700 48x25), "Base 4"
        toggle StationVisualProgram.MagPos4
    Button (1025,700 48x25), "Base 5"
        toggle StationVisualProgram.MagPos5
    Button (1088,700 48x25), "Base 6"
        toggle StationVisualProgram.BasePos6
    Button (1150,700 48x25), "Base 7"
        toggle StationVisualProgram.BasePos7
    Label (610,359 268x30), "REJECTED :("
    Group (132,701 703x151)
        Textfield (197,0 260x46), "PLEASE NOTE!!"
        Textfield (51,48 589x52), "To Reset: First press STOP then RESET"
        Textfield (0,101 703x50), "Manual Control: Turn AUTO OFF then press START"
END_VISUALIZATION
